{attribute addProperty BoxType "EK1122-0000-0018"}
{attribute addProperty Id "Beckhoff_EL3xxx_0030sub_EK1100EK1100_179A0949162"}
{attribute addProperty CRC "2831672833"}
{attribute addProperty SizeInBites "16"}
{attribute addProperty SizeInBytes "2"}
TYPE Beckhoff_EL3xxx_0030EK1122_A8C7E601 EXTENDS EK1122_179A0949 :
STRUCT
	{attribute addProperty Name "Beckhoff_EL3xxx_0030sub_EK1100"}
	Beckhoff_EL3xxx_0030sub_EK1100 : EK1100_179A0949;
END_STRUCT
END_TYPE

(* stored: Version 1.2.0.0, ProductVersion 3.1.4024.9
   DUT Beckhoff_EL3xxx_0030EK1122_A8C7E601: Id {3d26f692-bcbe-4a4f-98d6-fe7d4983e333} *)
